FUNCTION_BLOCK TC_OutputMapping (* Service Interface Function Block Type *)
  (* Standard: ISO 11783-10; Function: All Outputs; Type: TC according to ISO 11783-10; Description: Copyright (c) 2018, 2023 Jose Cabral, HR Agrartechnik GmbH This program and the accompanying materials are made available under the terms of the Eclipse Public License 2.0 which is available at https://www.eclipse.org/legal/epl-2.0/ SPDX-License-Identifier: EPL-2.0 this maps to QD 32 bit Process Data (PD) *)
  (* Version 1.0, 2018-12-05, Jose Cabral *)
  (* Version 1.1, 2022-08-04, Franz Höpfinger, HR Agrartechnik GmbH *)
  (* Version 1.2, 2023-01-05, Franz Höpfinger, HR Agrartechnik GmbH *)
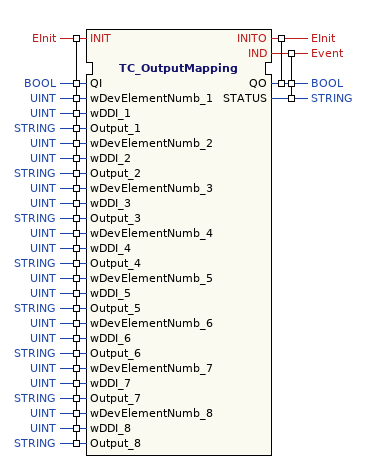
  EVENT_INPUT
    INIT : EInit WITH QI, wDevElementNumb_1, wDDI_1, Output_1, wDevElementNumb_2, wDDI_2, Output_2, wDevElementNumb_3, wDDI_3, Output_3, wDevElementNumb_4, wDDI_4, Output_4, wDevElementNumb_5, wDDI_5, Output_5, wDevElementNumb_6, wDDI_6, Output_6, wDevElementNumb_7, wDDI_7, Output_7, wDevElementNumb_8, wDDI_8, Output_8; (* Service Initialization *)
  END_EVENT
  EVENT_OUTPUT
    INITO : EInit WITH QO; (* Initialization Confirm *)
    IND WITH QO, STATUS; (* Indication from Resource *)
  END_EVENT
  VAR_INPUT
    QI : BOOL; (* Event Input Qualifier *)
    wDevElementNumb_1 : UINT; (* Requested element number of TC of Output 1 *)
    wDDI_1 : UINT; (* Data dictionary identifier of Output 1 *)
    Output_1 : STRING; (* Identifier for Output 1 *)
    wDevElementNumb_2 : UINT; (* Requested element number of TC of Output 2 *)
    wDDI_2 : UINT; (* Data dictionary identifier of Output 2 *)
    Output_2 : STRING; (* Identifier for Output 2 *)
    wDevElementNumb_3 : UINT; (* Requested element number of TC of Output 3 *)
    wDDI_3 : UINT; (* Data dictionary identifier of Output 3 *)
    Output_3 : STRING; (* Identifier for Output 3 *)
    wDevElementNumb_4 : UINT; (* Requested element number of TC of Output 4 *)
    wDDI_4 : UINT; (* Data dictionary identifier of Output 4 *)
    Output_4 : STRING; (* Identifier for Output 4 *)
    wDevElementNumb_5 : UINT; (* Requested element number of TC of Output 5 *)
    wDDI_5 : UINT; (* Data dictionary identifier of Output 5 *)
    Output_5 : STRING; (* Identifier for Output 5 *)
    wDevElementNumb_6 : UINT; (* Requested element number of TC of Output 6 *)
    wDDI_6 : UINT; (* Data dictionary identifier of Output 6 *)
    Output_6 : STRING; (* Identifier for Output 6 *)
    wDevElementNumb_7 : UINT; (* Requested element number of TC of Output 7 *)
    wDDI_7 : UINT; (* Data dictionary identifier of Output 7 *)
    Output_7 : STRING; (* Identifier for Output 7 *)
    wDevElementNumb_8 : UINT; (* Requested element number of TC of Output 8 *)
    wDDI_8 : UINT; (* Data dictionary identifier of Output 8 *)
    Output_8 : STRING; (* Identifier for Output 8 *)
  END_VAR
  VAR_OUTPUT
    QO : BOOL; (* Event Output Qualifier *)
    STATUS : STRING; (* Service Status *)
  END_VAR
END_FUNCTION_BLOCK
